(* Schneider Machine Expert - Basic project counter and timer, file version 1.6.0.0 *)
(* ProjectInformations: Name=New project *)

HARDWARE
  Cpu 0: TM221CE16R
  EthernetConfiguration: NetworkName=M221, IpAllocationMode=FixedAddress, IpAddress=0.0.0.0, SubnetMask=0.0.0.0
  SerialLineConfiguration: Baud=Baud19200, Parity=ParityEven, DataBits=DataBits8, StopBits=StopBits1, PhysicalMedium=PhysicalMediumRs485, TransmissionMode=TransmissionModeModbusRtu, SlaveId=1, Addressing=SlaveAddressing
  MastTask: UsePeriodScanMode=false, PeriodScan=100
  FastTask: Period=255
  CpuBehavior: StartingMode=StartAsPreviousState, AutoSaveRamOnEeprom=true, WatchdogPeriod=250

SYMBOLS  (address, symbol, comment, settings)
  %TM0        [Preset=202]

POU New POU
  (* SectionNumber=1 *)

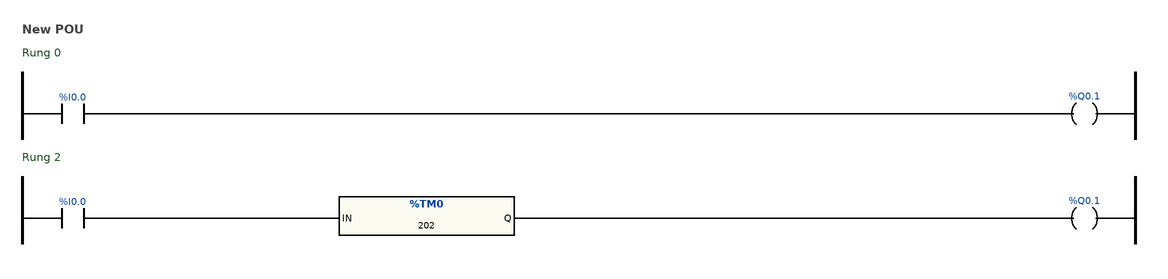

// Rung 0
  LD %I0.0
  ST %Q0.1
  // as ST:
  //   %Q0.1 := %I0.0;

// Rung 1
  BLK %C0
  LD %I0.0
  R
  LD %I0.0
  S
  LD %I0.0
  CU
  LD %I0.0
  CD
  OUT_BLK
  LD D
  ST %Q0.0
  END_BLK
  // as ST:
  //   %C0(R := %I0.0, S := %I0.0, CU := %I0.0, CD := %I0.0);
  //   %Q0.0 := %C0.D;

// Rung 2
  BLK %TM0
  LD %I0.0
  IN
  OUT_BLK
  LD Q
  ST %Q0.1
  END_BLK
  // as ST:
  //   %TM0(IN := %I0.0);
  //   %Q0.1 := %TM0.Q;
